(* IEC 61131-3 sources: stc/pkg/checker/testdata, 10 files *)

(* ---- fb_instance.st ---- *)
FUNCTION_BLOCK FB_Timer
VAR_INPUT
    enable : BOOL;
    preset : INT;
END_VAR
VAR_OUTPUT
    done : BOOL;
    elapsed : INT;
END_VAR
END_FUNCTION_BLOCK

PROGRAM Main
VAR
    timer1 : FB_Timer;
    result : BOOL;
    counter : INT;
END_VAR
    result := timer1.done;
    counter := timer1.elapsed;
END_PROGRAM

(* ---- forward_ref.st ---- *)
FUNCTION_BLOCK FB_Pump
VAR
    motor : FB_Motor;
END_VAR
END_FUNCTION_BLOCK

FUNCTION_BLOCK FB_Motor
VAR
    speed : INT;
END_VAR
END_FUNCTION_BLOCK

(* ---- forward_ref_members.st ---- *)
PROGRAM Main
VAR
    pump : FB_Pump;
    a : ST_A;
    t1 : T1;
    ta : TA;
    i : I_Motor;
    s : INT;
END_VAR
s := pump.motor.speed;
s := a.b.field;
t1 := s;
ta[0].field := s;
pump(cmd := TRUE);
END_PROGRAM

FUNCTION_BLOCK FB_Pump
VAR_INPUT
    cmd : BOOL;
END_VAR
VAR_OUTPUT
    motor : FB_Motor;
END_VAR
END_FUNCTION_BLOCK

FUNCTION_BLOCK FB_Motor
VAR_OUTPUT
    speed : INT;
END_VAR
END_FUNCTION_BLOCK

TYPE ST_A :
STRUCT
    b : ST_B;
END_STRUCT
END_TYPE

TYPE ST_B :
STRUCT
    field : INT;
END_STRUCT
END_TYPE

TYPE T1 : T2; END_TYPE

TYPE T2 : INT; END_TYPE

TYPE TA : ARRAY[0..1] OF ST_B; END_TYPE

INTERFACE I_Motor
END_INTERFACE

(* ---- vendor_oop.st ---- *)
FUNCTION_BLOCK MyFB
VAR
    counter : INT;
END_VAR

METHOD PUBLIC DoWork : BOOL
VAR_INPUT
    value : INT;
END_VAR
    DoWork := value > 0;
END_METHOD

END_FUNCTION_BLOCK

INTERFACE IRunnable
    METHOD Run : BOOL
    END_METHOD
END_INTERFACE

(* ---- array_struct.st ---- *)
PROGRAM Main
VAR
    arr : ARRAY[0..9] OF INT;
    idx : INT;
    val : INT;
    pt : S_Point;
    px : REAL;
END_VAR
    val := arr[idx];
    px := pt.x;
END_PROGRAM

(* ---- type_mismatch.st ---- *)
PROGRAM Main
VAR
    x : INT;
    y : STRING;
END_VAR
    x := y;
END_PROGRAM

(* ---- undeclared.st ---- *)
PROGRAM Main
VAR
    x : INT;
END_VAR
    x := undeclared_var;
END_PROGRAM

(* ---- unreachable.st ---- *)
PROGRAM Main
VAR
    x : INT;
    y : INT;
END_VAR

x := 1;
RETURN;
y := 2;  (* This is unreachable *)

END_PROGRAM

(* ---- unused_var.st ---- *)
PROGRAM Main
VAR
    unusedLocal : INT;
    usedLocal : INT;
END_VAR
VAR_INPUT
    unusedInput : INT;  (* Should NOT trigger warning *)
END_VAR

usedLocal := 42;

END_PROGRAM

(* ---- valid_program.st ---- *)
PROGRAM Main
VAR
    x : INT;
    y : REAL;
    z : BOOL;
END_VAR
    x := 42;
    y := 3.14;
    z := TRUE;
END_PROGRAM
